// TIA Portal V17 export
// export: Created 2024-08-07T21:43:50.1345699Z, ExportSetting WithDefaults, DisplayName Totally Integrated Automation Portal, DisplayVersion V17 Update 7, DisplayName TIA Portal Openness, DisplayVersion V17 Update 7, DisplayName TIA Portal Version Control Interface, DisplayVersion V17, DisplayName SINAMICS Startdrive Advanced, DisplayVersion V17 SP2, DisplayName SINAMICS Startdrive G110M, G120, G120C, G120D, G120P, G115D, DisplayVersion V17 SP2, DisplayName SINAMICS Startdrive G130, G150, S120, S150, SINAMICS MV, S210, DisplayVersion V17 SP2, DisplayName STEP 7 Professional, DisplayVersion V17 Update 7, DisplayName STEP 7 Safety, DisplayVersion V17 Update 6, DisplayName WinCC Advanced / Unified PC, DisplayVersion V17 Update 7
FUNCTION_BLOCK "FB_Devices"   // FB5100, LAD
{ S7_Optimized_Access := 'TRUE' }
VERSION : 0.1
// stored: AutoNumber false, IsIECCheckEnabled false, IsRetainMemResEnabled false, MemoryReserve 100, SetENOAutomatically false, UDAEnableTagReadback false
   VAR
      ServiceDoors_Instance_1 { S7_SetPoint := 'True'} : "serviceDoor";
      ServiceDoors_Instance_2 { S7_SetPoint := 'True'} : "serviceDoor";
      R_TRIG_Instance { S7_SetPoint := 'True'} : R_TRIG;
      HydraulicActive { S7_SetPoint := 'True'} : Bool;
      HydraulicActiveOffMem : Bool;
      HydraulicOnMem : Bool;
      IEC_Timer_0_Instance { S7_SetPoint := 'True'} : TON_TIME;
      IEC_Timer_0_Instance_1 { S7_SetPoint := 'True'} : TON_TIME;
      FB_TurnTable_Instance { S7_SetPoint := 'True'} : "FB_TurnTable";
      F_TRIG_Instance { S7_SetPoint := 'True'} : F_TRIG;
      edges { S7_SetPoint := 'True'} : Array[1..6] of Bool;
      ManualCommandOld : Int;
      R_TRIG_Instance_1 { S7_SetPoint := 'True'} : R_TRIG;
      R_TRIG_Instance_2 { S7_SetPoint := 'True'} : R_TRIG;
      R_TRIG_Instance_3 { S7_SetPoint := 'True'} : R_TRIG;
      R_TRIG_Instance_4 { S7_SetPoint := 'True'} : R_TRIG;
      R_TRIG_Instance_6 { S7_SetPoint := 'True'} : R_TRIG;
      R_TRIG_Instance_7 { S7_SetPoint := 'True'} : R_TRIG;
      R_TRIG_Instance_8 { S7_SetPoint := 'True'} : R_TRIG;
      R_TRIG_Instance_5 { S7_SetPoint := 'True'} : R_TRIG;
      edgesFitting : Array[1..4] of Bool;
      R_TRIG_V240Wp { S7_SetPoint := 'True'} : R_TRIG;
      R_TRIG_V240Bp { S7_SetPoint := 'True'} : R_TRIG;
      ReaderKeyence_Instance { S7_SetPoint := 'True'} : "ReaderKeyence";
      IEC_Timer_0_Instance_2 { S7_SetPoint := 'True'} : TON_TIME;
      FriedrichUnit1_Instance { S7_SetPoint := 'True'} : "FriedrichUnit";
      FriedrichUnit2_Instance { S7_SetPoint := 'True'} : "FriedrichUnit";
      Trig1 { S7_SetPoint := 'True'} : R_TRIG;
      Trig2 { S7_SetPoint := 'True'} : R_TRIG;
      Trig3 { S7_SetPoint := 'True'} : R_TRIG;
      Trig4 { S7_SetPoint := 'True'} : R_TRIG;
      Camera_CAM1 { S7_SetPoint := 'True'} : "Camera";
      Camera_CAM2 { S7_SetPoint := 'True'} : "Camera";
      Camera_CAM3 { S7_SetPoint := 'True'} : "Camera";
      Camera_CAM4 { S7_SetPoint := 'True'} : "Camera";
      RivetingCycleLeft_Instance { S7_SetPoint := 'True'} : "RivetingCycle";
      RivetingCycleRight_Instance { S7_SetPoint := 'True'} : "RivetingCycle";
   END_VAR
   VAR_TEMP
      posTemp : "UDT_PositionData";
      i : Int;
   END_VAR
   VAR_TEMP   // added for the SCL form of the ladder/FBD networks
      _w1 : Bool;
      _w2 : Bool;
      _w3 : Bool;
   END_VAR
BEGIN

REGION Network 1: Diagnostic fieldbus devices
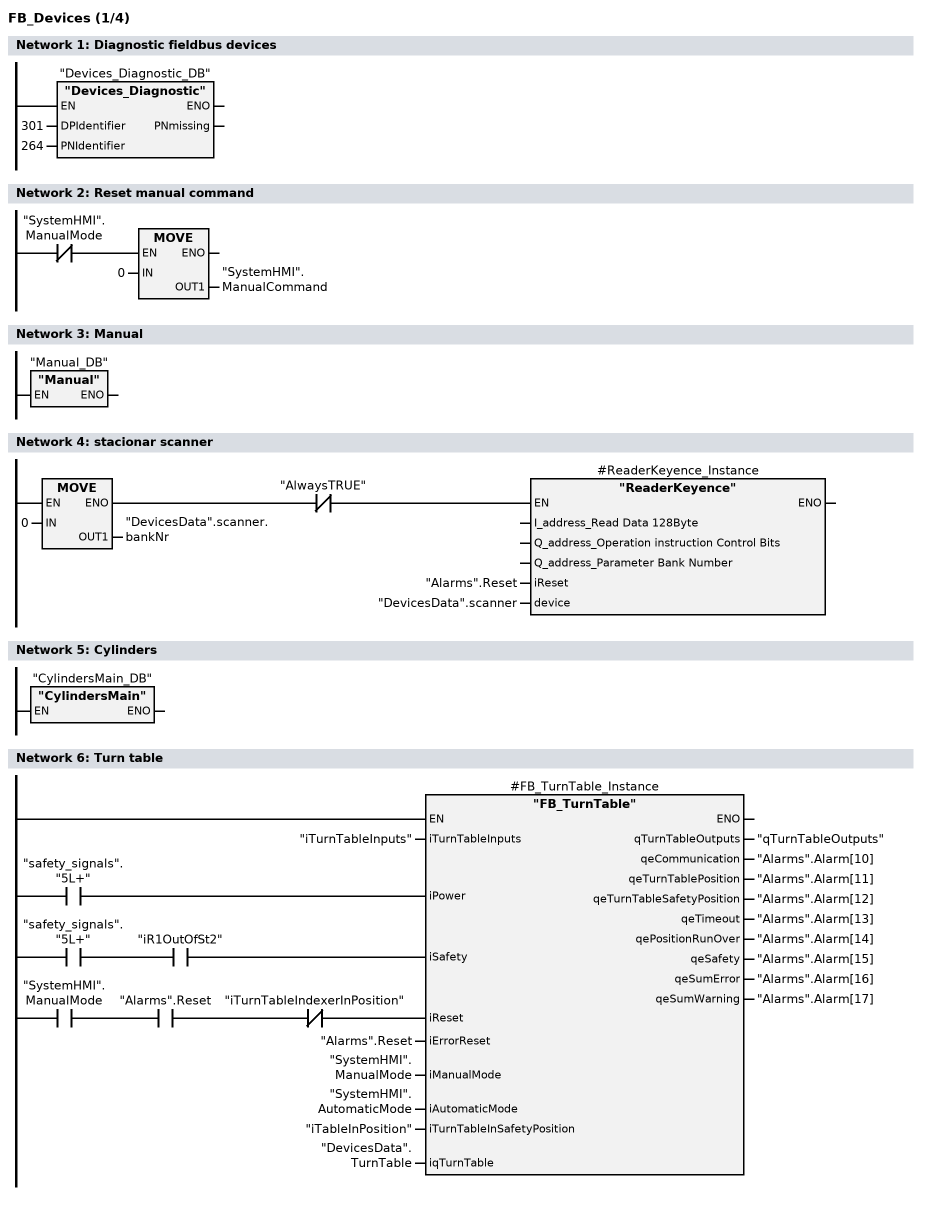
   RUNG wire#powerrail
      "Devices_Diagnostic_DB"(DPIdentifier := 301, PNIdentifier := 264, PNmissing =>)
   END_RUNG
   // the same network as SCL:
   "Devices_Diagnostic_DB"(DPIdentifier := 301, PNIdentifier := 264);   // "Devices_Diagnostic"
END_REGION

REGION Network 2: Reset manual command
   RUNG wire#powerrail
      I_Contact( "SystemHMI".ManualMode )
      Move(in := 0, out1 => "SystemHMI".ManualCommand)
   END_RUNG
   // the same network as SCL:
   IF NOT "SystemHMI".ManualMode THEN "SystemHMI".ManualCommand := 0; END_IF;
END_REGION

REGION Network 3: Manual
   RUNG wire#powerrail
      "Manual_DB"()
   END_RUNG
   // the same network as SCL:
   "Manual_DB"();   // "Manual"
END_REGION

REGION Network 4: stacionar scanner
   RUNG wire#powerrail
      Move(in := 0, out1 => "DevicesData".scanner.bankNr)
      I_Contact( "AlwaysTRUE" )
      #ReaderKeyence_Instance("I_address_Read Data 128Byte" :=, "Q_address_Operation instruction Control Bits" :=, "Q_address_Parameter Bank Number" :=, iReset := "Alarms".Reset, device := "DevicesData".scanner)
   END_RUNG
   // the same network as SCL:
   "DevicesData".scanner.bankNr := 0;
   IF NOT "AlwaysTRUE" THEN
       #ReaderKeyence_Instance(iReset := "Alarms".Reset, device := "DevicesData".scanner);   // "ReaderKeyence"
   END_IF;
END_REGION

REGION Network 5: Cylinders
   RUNG wire#powerrail
      "CylindersMain_DB"()
   END_RUNG
   // the same network as SCL:
   "CylindersMain_DB"();   // "CylindersMain"
END_REGION

REGION Network 6: Turn table
   RUNG wire#powerrail
      #FB_TurnTable_Instance(iPower := wire#w1, iSafety := wire#w2, iReset := wire#w3, iTurnTableInputs := "iTurnTableInputs", iErrorReset := "Alarms".Reset, iManualMode := "SystemHMI".ManualMode, iAutomaticMode := "SystemHMI".AutomaticMode, iTurnTableInSafetyPosition := "iTableInPosition", iqTurnTable := "DevicesData".TurnTable, qTurnTableOutputs => "qTurnTableOutputs", qeCommunication => "Alarms".Alarm[10], qeTurnTablePosition => "Alarms".Alarm[11], qeTurnTableSafetyPosition => "Alarms".Alarm[12], qeTimeout => "Alarms".Alarm[13], qePositionRunOver => "Alarms".Alarm[14], qeSafety => "Alarms".Alarm[15], qeSumError => "Alarms".Alarm[16], qeSumWarning => "Alarms".Alarm[17])
   END_RUNG
   RUNG wire#powerrail
      Contact( "safety_signals"."5L+" )
   END_RUNG wire#w1
   RUNG wire#powerrail
      Contact( "safety_signals"."5L+" )
      Contact( "iR1OutOfSt2" )
   END_RUNG wire#w2
   RUNG wire#powerrail
      Contact( "SystemHMI".ManualMode )
      Contact( "Alarms".Reset )
      I_Contact( "iTurnTableIndexerInPosition" )
   END_RUNG wire#w3
   // the same network as SCL:
   #FB_TurnTable_Instance(iTurnTableInputs := "iTurnTableInputs",   // "FB_TurnTable"
                          iPower := "safety_signals"."5L+",
                          iSafety := "safety_signals"."5L+" AND "iR1OutOfSt2",
                          iReset := "SystemHMI".ManualMode AND "Alarms".Reset AND NOT "iTurnTableIndexerInPosition",
                          iErrorReset := "Alarms".Reset,
                          iManualMode := "SystemHMI".ManualMode,
                          iAutomaticMode := "SystemHMI".AutomaticMode,
                          iTurnTableInSafetyPosition := "iTableInPosition",
                          iqTurnTable := "DevicesData".TurnTable,
                          qTurnTableOutputs => "qTurnTableOutputs",
                          qeCommunication => "Alarms".Alarm[10],
                          qeTurnTablePosition => "Alarms".Alarm[11],
                          qeTurnTableSafetyPosition => "Alarms".Alarm[12],
                          qeTimeout => "Alarms".Alarm[13],
                          qePositionRunOver => "Alarms".Alarm[14],
                          qeSafety => "Alarms".Alarm[15],
                          qeSumError => "Alarms".Alarm[16],
                          qeSumWarning => "Alarms".Alarm[17]);
END_REGION

REGION Network 7: Handle table positions
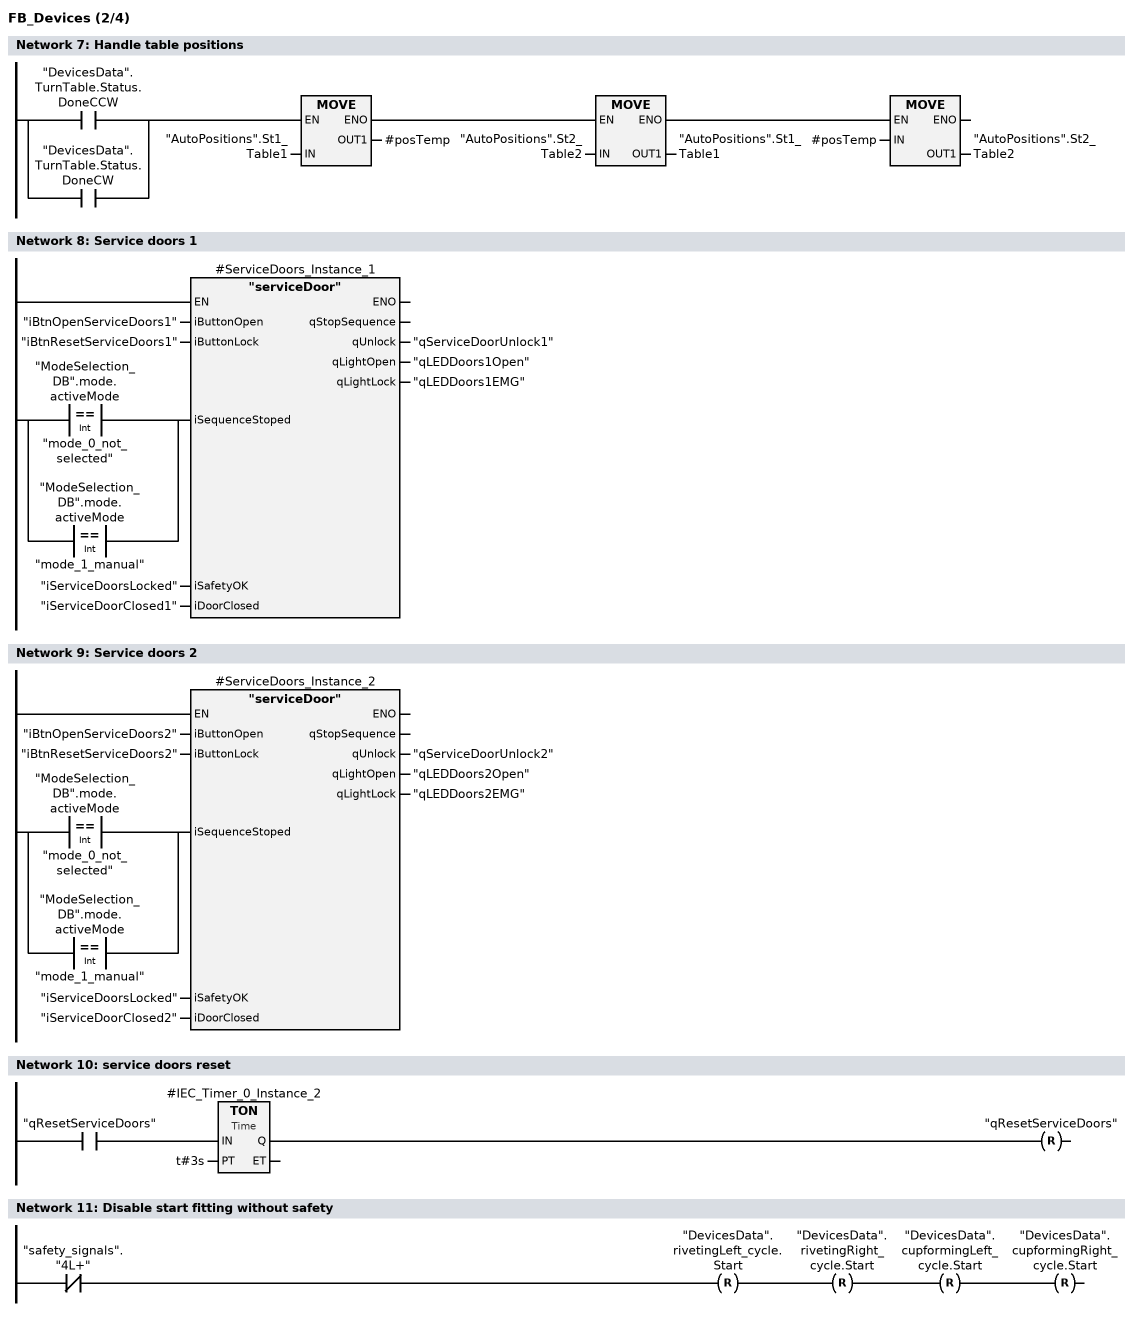
   RUNG wire#powerrail
      Contact( "DevicesData".TurnTable.Status.DoneCCW )
      wire#w1
      Move(in := "AutoPositions".St1_Table1, out1 => #posTemp)
      Move(in := "AutoPositions".St2_Table2, out1 => "AutoPositions".St1_Table1)
      Move(in := #posTemp, out1 => "AutoPositions".St2_Table2)
   END_RUNG
   RUNG wire#powerrail
      Contact( "DevicesData".TurnTable.Status.DoneCW )
   END_RUNG wire#w1
   // the same network as SCL:
   IF "DevicesData".TurnTable.Status.DoneCCW OR "DevicesData".TurnTable.Status.DoneCW THEN
       #posTemp := "AutoPositions".St1_Table1;
       "AutoPositions".St1_Table1 := "AutoPositions".St2_Table2;
       "AutoPositions".St2_Table2 := #posTemp;
   END_IF;
END_REGION

REGION Network 8: Service doors 1
   RUNG wire#powerrail
      #ServiceDoors_Instance_1(iSequenceStoped := wire#w1, iButtonOpen := "iBtnOpenServiceDoors1", iButtonLock := "iBtnResetServiceDoors1", iSafetyOK := "iServiceDoorsLocked", iDoorClosed := "iServiceDoorClosed1", qStopSequence =>, qUnlock => "qServiceDoorUnlock1", qLightOpen => "qLEDDoors1Open", qLightLock => "qLEDDoors1EMG")
   END_RUNG
   RUNG wire#powerrail
      { S7_Templates := "SrcType := Int" } EQ_Contact(in1 := "ModeSelection_DB".mode.activeMode, in2 := "mode_0_not_selected")
   END_RUNG wire#w1
   RUNG wire#powerrail
      { S7_Templates := "SrcType := Int" } EQ_Contact(in1 := "ModeSelection_DB".mode.activeMode, in2 := "mode_1_manual")
   END_RUNG wire#w1
   // the same network as SCL:
   #ServiceDoors_Instance_1(iButtonOpen := "iBtnOpenServiceDoors1",   // "serviceDoor"
                           iButtonLock := "iBtnResetServiceDoors1",
                           iSequenceStoped := ("ModeSelection_DB".mode.activeMode = "mode_0_not_selected") OR ("ModeSelection_DB".mode.activeMode = "mode_1_manual"),
                           iSafetyOK := "iServiceDoorsLocked",
                           iDoorClosed := "iServiceDoorClosed1",
                           qUnlock => "qServiceDoorUnlock1",
                           qLightOpen => "qLEDDoors1Open",
                           qLightLock => "qLEDDoors1EMG");
END_REGION

REGION Network 9: Service doors 2
   RUNG wire#powerrail
      #ServiceDoors_Instance_2(iSequenceStoped := wire#w1, iButtonOpen := "iBtnOpenServiceDoors2", iButtonLock := "iBtnResetServiceDoors2", iSafetyOK := "iServiceDoorsLocked", iDoorClosed := "iServiceDoorClosed2", qStopSequence =>, qUnlock => "qServiceDoorUnlock2", qLightOpen => "qLEDDoors2Open", qLightLock => "qLEDDoors2EMG")
   END_RUNG
   RUNG wire#powerrail
      { S7_Templates := "SrcType := Int" } EQ_Contact(in1 := "ModeSelection_DB".mode.activeMode, in2 := "mode_0_not_selected")
   END_RUNG wire#w1
   RUNG wire#powerrail
      { S7_Templates := "SrcType := Int" } EQ_Contact(in1 := "ModeSelection_DB".mode.activeMode, in2 := "mode_1_manual")
   END_RUNG wire#w1
   // the same network as SCL:
   #ServiceDoors_Instance_2(iButtonOpen := "iBtnOpenServiceDoors2",   // "serviceDoor"
                           iButtonLock := "iBtnResetServiceDoors2",
                           iSequenceStoped := ("ModeSelection_DB".mode.activeMode = "mode_0_not_selected") OR ("ModeSelection_DB".mode.activeMode = "mode_1_manual"),
                           iSafetyOK := "iServiceDoorsLocked",
                           iDoorClosed := "iServiceDoorClosed2",
                           qUnlock => "qServiceDoorUnlock2",
                           qLightOpen => "qLEDDoors2Open",
                           qLightLock => "qLEDDoors2EMG");
END_REGION

REGION Network 10: service doors reset
   RUNG wire#powerrail
      Contact( "qResetServiceDoors" )
      { S7_Templates := "time_type := Time" } #IEC_Timer_0_Instance_2.TON(pt := t#3s, et =>)
      R_Coil( "qResetServiceDoors" )
   END_RUNG
   // the same network as SCL:
   #IEC_Timer_0_Instance_2(IN := "qResetServiceDoors", PT := t#3s);   // TON
   IF #IEC_Timer_0_Instance_2.Q THEN "qResetServiceDoors" := FALSE; END_IF;
END_REGION

REGION Network 11: Disable start fitting without safety
   RUNG wire#powerrail
      I_Contact( "safety_signals"."4L+" )
      R_Coil( "DevicesData".rivetingLeft_cycle.Start )
      R_Coil( "DevicesData".rivetingRight_cycle.Start )
      R_Coil( "DevicesData".cupformingLeft_cycle.Start )
      R_Coil( "DevicesData".cupformingRight_cycle.Start )
   END_RUNG
   // the same network as SCL:
   IF NOT "safety_signals"."4L+" THEN
       "DevicesData".rivetingLeft_cycle.Start := FALSE;
       "DevicesData".rivetingRight_cycle.Start := FALSE;
       "DevicesData".cupformingLeft_cycle.Start := FALSE;
       "DevicesData".cupformingRight_cycle.Start := FALSE;
   END_IF;
END_REGION

REGION Network 12: Fittings - Cyle times measurement
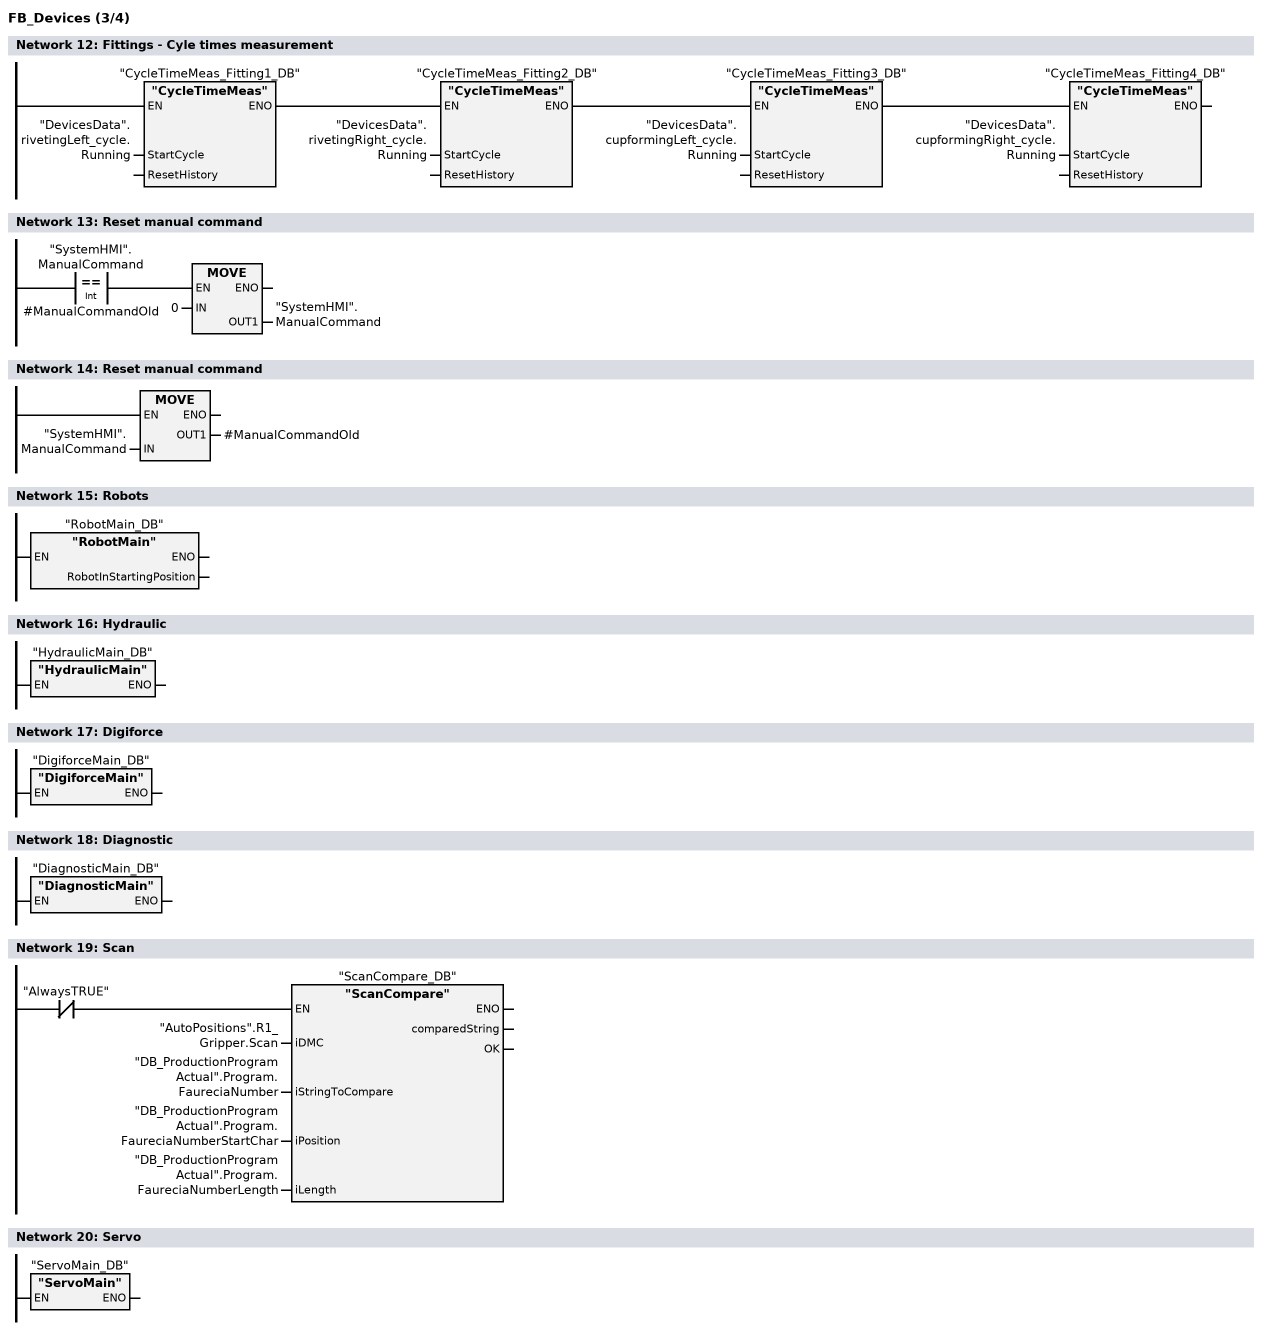
   RUNG wire#powerrail
      "CycleTimeMeas_Fitting1_DB"(StartCycle := "DevicesData".rivetingLeft_cycle.Running, ResetHistory :=)
      "CycleTimeMeas_Fitting2_DB"(StartCycle := "DevicesData".rivetingRight_cycle.Running, ResetHistory :=)
      "CycleTimeMeas_Fitting3_DB"(StartCycle := "DevicesData".cupformingLeft_cycle.Running, ResetHistory :=)
      "CycleTimeMeas_Fitting4_DB"(StartCycle := "DevicesData".cupformingRight_cycle.Running, ResetHistory :=)
   END_RUNG
   // the same network as SCL:
   "CycleTimeMeas_Fitting1_DB"(StartCycle := "DevicesData".rivetingLeft_cycle.Running, ENO => #_w1);   // "CycleTimeMeas"
   "CycleTimeMeas_Fitting2_DB"(EN := #_w1, StartCycle := "DevicesData".rivetingRight_cycle.Running, ENO => #_w2);   // "CycleTimeMeas"
   "CycleTimeMeas_Fitting3_DB"(EN := #_w2,   // "CycleTimeMeas"
                           StartCycle := "DevicesData".cupformingLeft_cycle.Running,
                           ENO => #_w3);
   IF #_w3 THEN
       "CycleTimeMeas_Fitting4_DB"(StartCycle := "DevicesData".cupformingRight_cycle.Running);   // "CycleTimeMeas"
   END_IF;
END_REGION

REGION Network 13: Reset manual command
   RUNG wire#powerrail
      { S7_Templates := "SrcType := Int" } EQ_Contact(in1 := "SystemHMI".ManualCommand, in2 := #ManualCommandOld)
      Move(in := 0, out1 => "SystemHMI".ManualCommand)
   END_RUNG
   // the same network as SCL:
   IF "SystemHMI".ManualCommand = #ManualCommandOld THEN "SystemHMI".ManualCommand := 0; END_IF;
END_REGION

REGION Network 14: Reset manual command
   RUNG wire#powerrail
      Move(in := "SystemHMI".ManualCommand, out1 => #ManualCommandOld)
   END_RUNG
   // the same network as SCL:
   #ManualCommandOld := "SystemHMI".ManualCommand;
END_REGION

REGION Network 15: Robots
   RUNG wire#powerrail
      "RobotMain_DB"(RobotInStartingPosition =>)
   END_RUNG
   // the same network as SCL:
   "RobotMain_DB"();   // "RobotMain"
END_REGION

REGION Network 16: Hydraulic
   RUNG wire#powerrail
      "HydraulicMain_DB"()
   END_RUNG
   // the same network as SCL:
   "HydraulicMain_DB"();   // "HydraulicMain"
END_REGION

REGION Network 17: Digiforce
   RUNG wire#powerrail
      "DigiforceMain_DB"()
   END_RUNG
   // the same network as SCL:
   "DigiforceMain_DB"();   // "DigiforceMain"
END_REGION

REGION Network 18: Diagnostic
   RUNG wire#powerrail
      "DiagnosticMain_DB"()
   END_RUNG
   // the same network as SCL:
   "DiagnosticMain_DB"();   // "DiagnosticMain"
END_REGION

REGION Network 19: Scan
   RUNG wire#powerrail
      I_Contact( "AlwaysTRUE" )
      "ScanCompare_DB"(iDMC := "AutoPositions".R1_Gripper.Scan, iStringToCompare := "DB_ProductionProgramActual".Program.FaureciaNumber, iPosition := "DB_ProductionProgramActual".Program.FaureciaNumberStartChar, iLength := "DB_ProductionProgramActual".Program.FaureciaNumberLength, comparedString =>, OK =>)
   END_RUNG
   // the same network as SCL:
   IF NOT "AlwaysTRUE" THEN
       "ScanCompare_DB"(iDMC := "AutoPositions".R1_Gripper.Scan,   // "ScanCompare"
                        iStringToCompare := "DB_ProductionProgramActual".Program.FaureciaNumber,
                        iPosition := "DB_ProductionProgramActual".Program.FaureciaNumberStartChar,
                        iLength := "DB_ProductionProgramActual".Program.FaureciaNumberLength);
   END_IF;
END_REGION

REGION Network 20: Servo
   RUNG wire#powerrail
      "ServoMain_DB"()
   END_RUNG
   // the same network as SCL:
   "ServoMain_DB"();   // "ServoMain"
END_REGION

REGION Network 21 (SCL): Friedrich1 R
   IF "HMIData".ManualCommand = 611 THEN
       "DevicesData".Friedrich1.Start := true;
   END_IF;

   #FriedrichUnit1_Instance(safetyOK := "safety_signals"."4L+",
                            iReady := "iRivetingReady1",
                            iZ1OK := "iRivetingZ1ok1",
                            iH1OK := "iRivetingH1ok1",
                            iH2OK := "iRivetingH2ok1",
                            iTimeOK := "iRivetingTimeOk1",
                            iNoAlarm := "iRivetingNoError1",
                            FriedrichNumber := 1,
                            Port := 39000,
                            IP1 := 192,
                            IP2 := 168,
                            IP3 := 16,
                            IP4 := 43,
                            ID := 2,
                            qStart => "qRiveting1Start",
                            qPrgbit4 => "qRiveting1Bit4",
                            qPrgbit3 => "qRiveting1Bit3",
                            qPrgbit2 => "qRiveting1Bit2",
                            qPrgbit1 => "qRiveting1Bit1",
                            qPrgbit0 => "qRiveting1Bit0",
                            RivetData := "DevicesData".Friedrich1);
   "qFriedrich1_setup_mode" := "DB_MainData".MachineMode <> 2 AND "DB_MainData".MachineMode <> 3;

   #Trig1(CLK:="DevicesData".Friedrich1.OK);
   #Trig2(CLK:="DevicesData".Friedrich1.NOK);
   "RivetingHistoryRight_DB"(iNewCycle := #Trig1.Q OR #Trig2.Q,
                             iData := "DevicesData".Friedrich1);

   #RivetingCycleRight_Instance(parameters := "DB_ProductionProgramActual".Program.Riveting_program_right,
                                basicPosition := "DevicesData".Friedrich1.Ready AND "DevicesData".Cylinders[MM340_RivetingUnitRight].InBp AND "DevicesData".Cylinders[MM344_RivetingSupportRight].InBp,
                                twoRivets := "DB_ProductionProgramActual".Program.Total_number_of_rivets_4,
                                MeasuredData1=>"AutoInfo".PartMeasuredData.RightRiveting1,
                                MeasuredData2=>"AutoInfo".PartMeasuredData.RightRiveting2,
                                riveter := "DevicesData".Friedrich1,
                                data := "DevicesData".rivetingRight_cycle,
                                cylinderSupport := "DevicesData".Cylinders[MM344_RivetingSupportRight],
                                cylinderShift := "DevicesData".Cylinders[MM340_RivetingUnitRight]);
END_REGION

REGION Network 22 (SCL): Friedrich2 L
   IF "HMIData".ManualCommand = 612 THEN
       "DevicesData".Friedrich2.Start := true;
   END_IF;
   #FriedrichUnit2_Instance(safetyOK := "safety_signals"."4L+",
                            iReady := "iRivetingReady2",
                            iZ1OK := "iRivetingZ1ok2",
                            iH1OK := "iRivetingH1ok2",
                            iH2OK := "iRivetingH2ok2",
                            iTimeOK := "iRivetingTimeOk2",
                            iNoAlarm := "iRivetingNoError2",
                            FriedrichNumber := 2,
                            Port := 39000,
                            IP1 := 192,
                            IP2 := 168,
                            IP3 := 16,
                            IP4 := 44,
                            ID := 3,
                            qStart => "qRiveting2Start",
                            qPrgbit4 => "qRiveting2Bit4",
                            qPrgbit3 => "qRiveting2Bit3",
                            qPrgbit2 => "qRiveting2Bit2",
                            qPrgbit1 => "qRiveting2Bit1",
                            qPrgbit0 => "qRiveting2Bit0",
                            RivetData := "DevicesData".Friedrich2);
   "qFriedrich2_setup_mode" := "DB_MainData".MachineMode <> 2 AND "DB_MainData".MachineMode <> 3;

   #Trig3(CLK:="DevicesData".Friedrich2.OK);
   #Trig4(CLK:="DevicesData".Friedrich2.NOK);
   "RivetingHistoryLeft_DB"(iNewCycle := #Trig3.Q OR #Trig4.Q,
                            iData := "DevicesData".Friedrich2);

   #RivetingCycleLeft_Instance(parameters := "DB_ProductionProgramActual".Program.Riveting_program_left,
                               basicPosition := "DevicesData".Friedrich2.Ready AND "DevicesData".Cylinders[MM342_RivetingUnitLeft].InBp AND "DevicesData".Cylinders[MM346_RivetingSupportLeft].InBp,
                               twoRivets := "DB_ProductionProgramActual".Program.Total_number_of_rivets_4,
                               MeasuredData1=>"AutoInfo".PartMeasuredData.LeftRiveting1,
                               MeasuredData2=>"AutoInfo".PartMeasuredData.LeftRiveting2,
                               riveter := "DevicesData".Friedrich2,
                               data := "DevicesData".rivetingLeft_cycle,
                               cylinderSupport := "DevicesData".Cylinders[MM346_RivetingSupportLeft],
                               cylinderShift := "DevicesData".Cylinders[MM342_RivetingUnitLeft]);

   REGION cycles handshake
       IF "SystemHMI".AutomaticMode THEN
           IF "DevicesData".cupformingLeft_cycle.Done AND "DevicesData".cupformingRight_cycle.Done THEN
               "DevicesData".rivetingLeft_cycle.ContinueFitting := TRUE;
               "DevicesData".rivetingRight_cycle.ContinueFitting := TRUE;
           END_IF;
       END_IF;
       "DevicesData".rivetingLeft_cycle.ContinueFitting := TRUE;
       "DevicesData".rivetingRight_cycle.ContinueFitting := TRUE;

       IF "SystemHMI".ManualMode THEN
           "DevicesData".rivetingLeft_cycle.ContinueFitting := true;
           "DevicesData".rivetingRight_cycle.ContinueFitting := true;
       END_IF;
   END_REGION
END_REGION

REGION Network 23
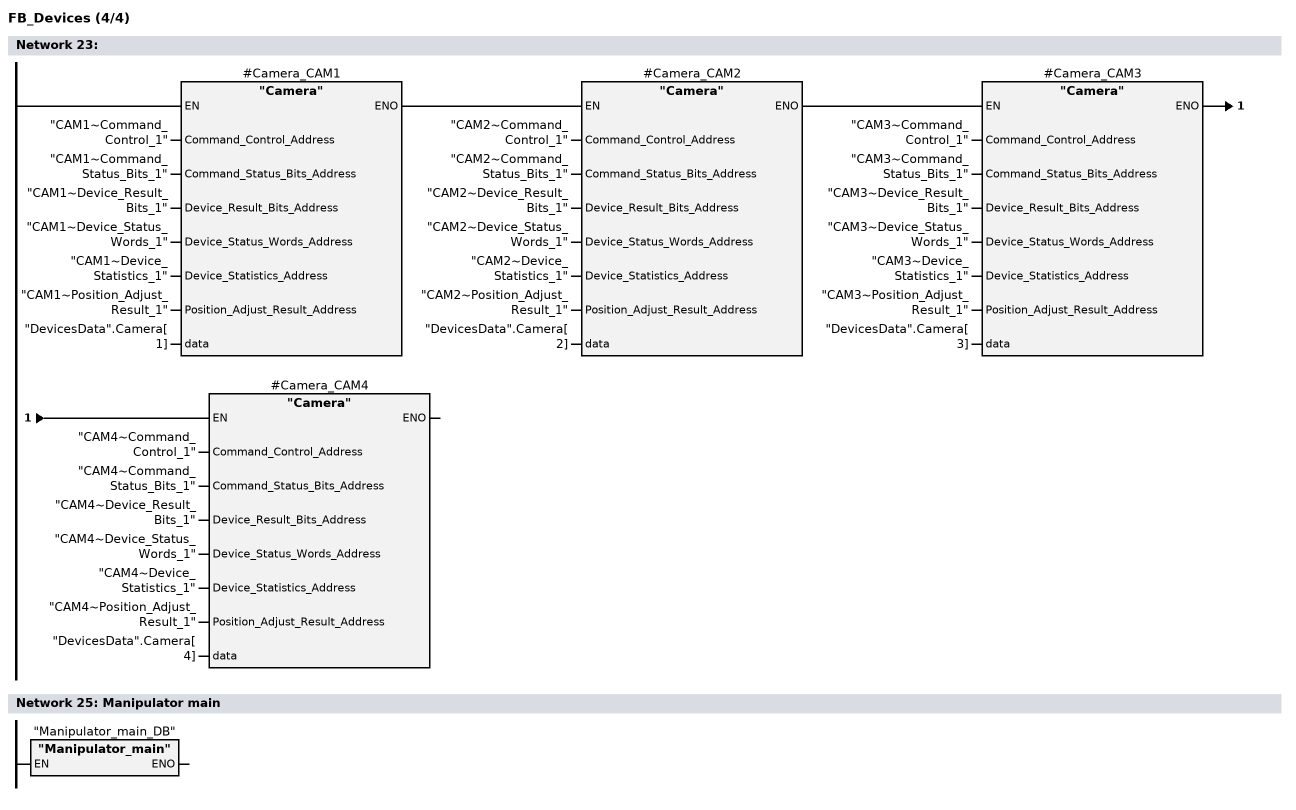
   RUNG wire#powerrail
      #Camera_CAM1(Command_Control_Address := "CAM1~Command_Control_1", Command_Status_Bits_Address := "CAM1~Command_Status_Bits_1", Device_Result_Bits_Address := "CAM1~Device_Result_Bits_1", Device_Status_Words_Address := "CAM1~Device_Status_Words_1", Device_Statistics_Address := "CAM1~Device_Statistics_1", Position_Adjust_Result_Address := "CAM1~Position_Adjust_Result_1", data := "DevicesData".Camera[1])
      #Camera_CAM2(Command_Control_Address := "CAM2~Command_Control_1", Command_Status_Bits_Address := "CAM2~Command_Status_Bits_1", Device_Result_Bits_Address := "CAM2~Device_Result_Bits_1", Device_Status_Words_Address := "CAM2~Device_Status_Words_1", Device_Statistics_Address := "CAM2~Device_Statistics_1", Position_Adjust_Result_Address := "CAM2~Position_Adjust_Result_1", data := "DevicesData".Camera[2])
      #Camera_CAM3(Command_Control_Address := "CAM3~Command_Control_1", Command_Status_Bits_Address := "CAM3~Command_Status_Bits_1", Device_Result_Bits_Address := "CAM3~Device_Result_Bits_1", Device_Status_Words_Address := "CAM3~Device_Status_Words_1", Device_Statistics_Address := "CAM3~Device_Statistics_1", Position_Adjust_Result_Address := "CAM3~Position_Adjust_Result_1", data := "DevicesData".Camera[3])
      #Camera_CAM4(Command_Control_Address := "CAM4~Command_Control_1", Command_Status_Bits_Address := "CAM4~Command_Status_Bits_1", Device_Result_Bits_Address := "CAM4~Device_Result_Bits_1", Device_Status_Words_Address := "CAM4~Device_Status_Words_1", Device_Statistics_Address := "CAM4~Device_Statistics_1", Position_Adjust_Result_Address := "CAM4~Position_Adjust_Result_1", data := "DevicesData".Camera[4])
   END_RUNG
   // the same network as SCL:
   #Camera_CAM1(Command_Control_Address := "CAM1~Command_Control_1",   // "Camera"
                Command_Status_Bits_Address := "CAM1~Command_Status_Bits_1",
                Device_Result_Bits_Address := "CAM1~Device_Result_Bits_1",
                Device_Status_Words_Address := "CAM1~Device_Status_Words_1",
                Device_Statistics_Address := "CAM1~Device_Statistics_1",
                Position_Adjust_Result_Address := "CAM1~Position_Adjust_Result_1",
                data := "DevicesData".Camera[1],
                ENO => #_w1);
   #Camera_CAM2(EN := #_w1,   // "Camera"
                Command_Control_Address := "CAM2~Command_Control_1",
                Command_Status_Bits_Address := "CAM2~Command_Status_Bits_1",
                Device_Result_Bits_Address := "CAM2~Device_Result_Bits_1",
                Device_Status_Words_Address := "CAM2~Device_Status_Words_1",
                Device_Statistics_Address := "CAM2~Device_Statistics_1",
                Position_Adjust_Result_Address := "CAM2~Position_Adjust_Result_1",
                data := "DevicesData".Camera[2],
                ENO => #_w2);
   #Camera_CAM3(EN := #_w2,   // "Camera"
                Command_Control_Address := "CAM3~Command_Control_1",
                Command_Status_Bits_Address := "CAM3~Command_Status_Bits_1",
                Device_Result_Bits_Address := "CAM3~Device_Result_Bits_1",
                Device_Status_Words_Address := "CAM3~Device_Status_Words_1",
                Device_Statistics_Address := "CAM3~Device_Statistics_1",
                Position_Adjust_Result_Address := "CAM3~Position_Adjust_Result_1",
                data := "DevicesData".Camera[3],
                ENO => #_w3);
   IF #_w3 THEN
       #Camera_CAM4(Command_Control_Address := "CAM4~Command_Control_1",   // "Camera"
                    Command_Status_Bits_Address := "CAM4~Command_Status_Bits_1",
                    Device_Result_Bits_Address := "CAM4~Device_Result_Bits_1",
                    Device_Status_Words_Address := "CAM4~Device_Status_Words_1",
                    Device_Statistics_Address := "CAM4~Device_Statistics_1",
                    Position_Adjust_Result_Address := "CAM4~Position_Adjust_Result_1",
                    data := "DevicesData".Camera[4]);
   END_IF;
END_REGION

REGION Network 24 (SCL)
   "DevicesData".Camera[1].ProgramNumber := USINT_TO_SINT("DB_ProductionProgramActual".Program.Camera_program[1]);
   "DevicesData".Camera[2].ProgramNumber := USINT_TO_SINT("DB_ProductionProgramActual".Program.Camera_program[2]);
   "DevicesData".Camera[3].ProgramNumber := USINT_TO_SINT("DB_ProductionProgramActual".Program.Camera_program[3]);
   "DevicesData".Camera[4].ProgramNumber := USINT_TO_SINT("DB_ProductionProgramActual".Program.Camera_program[4]);
END_REGION

REGION Network 25: Manipulator main
   RUNG wire#powerrail
      "Manipulator_main_DB"()
   END_RUNG
   // the same network as SCL:
   "Manipulator_main_DB"();   // "Manipulator_main"
END_REGION
END_FUNCTION_BLOCK
